Omron CX-Programmer project NewProject (CX-Programmer 9.73)

# PLC NewPLC1: CP1E N20

## Global symbols (name address type ; comment)
0.00 BOOL  ; suis
100.00 BOOL  ; lamp 1
100.02 BOOL  ; LAMP 3
100.07 BOOL  ; LAMP2
T002 BOOL  ; TIMER

## Program NewProgram1 (cyclic task 0)

### Section Section1

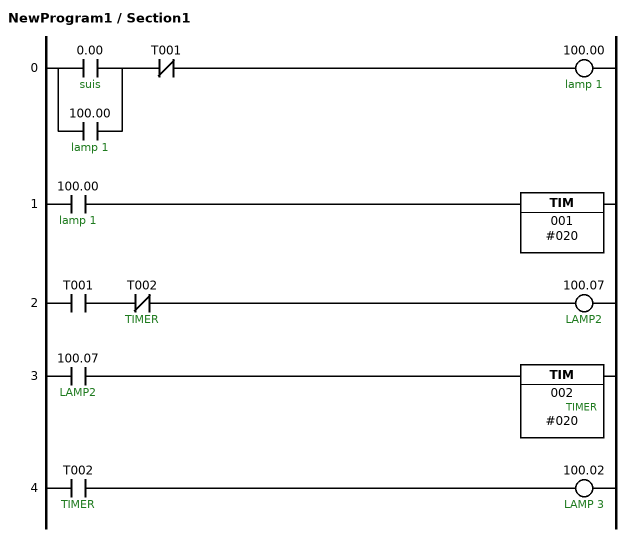
; rung 0
LD 0.00  ; suis
OR 100.00  ; lamp 1
ANDNOT T001
OUT 100.00  ; lamp 1
; rung 1
LD 100.00  ; lamp 1
TIM 001 #020
; rung 2
LD T001
ANDNOT T002  ; TIMER
OUT 100.07  ; LAMP2
; rung 3
LD 100.07  ; LAMP2
TIM 002 #020  ; TIMER
; rung 4
LD T002  ; TIMER
OUT 100.02  ; LAMP 3

### Section END
; rung 0
END(001)